LIN {X 0,Y 44.824,Z 368.173,A -85,B 0,C 180,E1 -30619.848,E2 -30619.848} C_VEL
LIN {X 0,Y 35.691,Z 373.226,A -85,B 0,C 180,E1 -30627.637,E2 -30627.637} C_VEL
LIN {X 0,Y 27.611,Z 377.135,A -85,B 0,C 180,E1 -30640.238,E2 -30640.238} C_VEL
LIN {X 0,Y 23.443,Z 379.156,A -85,B 0,C 180,E1 -30653.18,E2 -30653.18} C_VEL
LIN {X 0,Y 20.791,Z 380.755,A -85,B 0,C 180,E1 -30670.262,E2 -30670.262} C_VEL
LIN {X 0,Y 20.222,Z 381.925,A -85,B 0,C 180,E1 -30690.018,E2 -30690.018} C_VEL
LIN {X 0,Y 20.865,Z 382.602,A -85,B 0,C 180,E1 -30709.702,E2 -30709.702} C_VEL
LIN {X 0,Y 27.747,Z 382.794,A -85,B 0,C 180,E1 -30739.472,E2 -30739.472} C_VEL
LIN {X 0,Y 32.934,Z 382.312,A -85,B 0,C 180,E1 -30748.624,E2 -30748.624} C_VEL
LIN {X 0,Y 44.972,Z 380.11,A -85,B 0,C 180,E1 -30759.681,E2 -30759.681} C_VEL
LIN {X 0,Y 55.869,Z 376.992,A -85,B 0,C 180,E1 -30765.188,E2 -30765.188} C_VEL
LIN {X 0,Y 67.983,Z 372.218,A -85,B 0,C 180,E1 -30769.165,E2 -30769.165} C_VEL
LIN {X 0,Y 79.908,Z 365.993,A -85,B 0,C 180,E1 -30771.694,E2 -30771.694} C_VEL
LIN {X 0,Y 90.237,Z 359.24,A -85,B 0,C 180,E1 -30773.253,E2 -30773.253} C_VEL
LIN {X 0,Y 100.625,Z 350.879,A -85,B 0,C 180,E1 -30774.452,E2 -30774.452} C_VEL
LIN {X 0,Y 109.319,Z 342.285,A -85,B 0,C 180,E1 -30775.22,E2 -30775.22} C_VEL
LIN {X 0,Y 118.031,Z 331.706,A -85,B 0,C 180,E1 -30775.863,E2 -30775.863} C_VEL
LIN {X 0,Y 125.022,Z 321.224,A -85,B 0,C 180,E1 -30776.229,E2 -30776.229} C_VEL
LIN {X 0,Y 130.54,Z 310.906,A -85,B 0,C 180,E1 -30776.572,E2 -30776.572} C_VEL
LIN {X 0,Y 132.33,Z 306.946,A -85,B 0,C 180,E1 -30776.668,E2 -30776.668} C_VEL
LIN {X 0,Y 133.078,Z 305.198,A -85,B 0,C 180,E1 -30776.973,E2 -30776.973} C_VEL
LIN {X 0,Y 133.057,Z 305.114,A -85,B 0,C 180,E1 -30778.892,E2 -30778.892} C_VEL
LIN {X 0,Y 132.222,Z 307.019,A -85,B 0,C 180,E1 -30779.287,E2 -30779.287} C_VEL
LIN {X 0,Y 126.51,Z 318.425,A -85,B 0,C 180,E1 -30779.775,E2 -30779.775} C_VEL
LIN {X 0,Y 119.485,Z 329.469,A -85,B 0,C 180,E1 -30780.49,E2 -30780.49} C_VEL
LIN {X 0,Y 110.727,Z 340.358,A -85,B 0,C 180,E1 -30781.354,E2 -30781.354} C_VEL
LIN {X 0,Y 102.002,Z 349.18,A -85,B 0,C 180,E1 -30782.415,E2 -30782.415} C_VEL
LIN {X 0,Y 93.311,Z 356.441,A -85,B 0,C 180,E1 -30783.608,E2 -30783.608} C_VEL
LIN {X 0,Y 82.961,Z 363.561,A -85,B 0,C 180,E1 -30785.466,E2 -30785.466} C_VEL
LIN {X 0,Y 74.417,Z 368.349,A -85,B 0,C 180,E1 -30787.386,E2 -30787.386} C_VEL
LIN {X 0,Y 64.274,Z 372.98,A -85,B 0,C 180,E1 -30790.205,E2 -30790.205} C_VEL
LIN {X 0,Y 54.138,Z 376.491,A -85,B 0,C 180,E1 -30794.071,E2 -30794.071} C_VEL
LIN {X 0,Y 44.695,Z 378.993,A -85,B 0,C 180,E1 -30799.336,E2 -30799.336} C_VEL
LIN {X 0,Y 38.582,Z 380.15,A -85,B 0,C 180,E1 -30804.365,E2 -30804.365} C_VEL
LIN {X 0,Y 28.683,Z 381.121,A -85,B 0,C 180,E1 -30818.204,E2 -30818.204} C_VEL
LIN {X 0,Y 24.447,Z 381.264,A -85,B 0,C 180,E1 -30827.11,E2 -30827.11} C_VEL
LIN {X 0,Y 17.613,Z 380.911,A -85,B 0,C 180,E1 -30847.022,E2 -30847.022} C_VEL
LIN {X 0,Y 14.511,Z 380.036,A -85,B 0,C 180,E1 -30873.529,E2 -30873.529} C_VEL
LIN {X 0,Y 15.348,Z 378.997,A -85,B 0,C 180,E1 -30896.007,E2 -30896.007} C_VEL
LIN {X 0,Y 16.29,Z 378.557,A -85,B 0,C 180,E1 -30902.168,E2 -30902.168} C_VEL
LIN {X 0,Y 25.335,Z 375.258,A -85,B 0,C 180,E1 -30926.3,E2 -30926.3} C_VEL
LIN {X 0,Y 34.603,Z 371.292,A -85,B 0,C 180,E1 -30936.032,E2 -30936.032} C_VEL
LIN {X 0,Y 44.392,Z 366.186,A -85,B 0,C 180,E1 -30941.757,E2 -30941.757} C_VEL
LIN {X 0,Y 54.436,Z 359.759,A -85,B 0,C 180,E1 -30945.504,E2 -30945.504} C_VEL
LIN {X 0,Y 64.618,Z 351.765,A -85,B 0,C 180,E1 -30948.167,E2 -30948.167} C_VEL
LIN {X 0,Y 73.179,Z 343.603,A -85,B 0,C 180,E1 -30949.832,E2 -30949.832} C_VEL
LIN {X 0,Y 81.775,Z 333.642,A -85,B 0,C 180,E1 -30951.209,E2 -30951.209} C_VEL
LIN {X 0,Y 89.521,Z 322.368,A -85,B 0,C 180,E1 -30952.335,E2 -30952.335} C_VEL
LIN {X 0,Y 95.579,Z 311.302,A -85,B 0,C 180,E1 -30953.017,E2 -30953.017} C_VEL
LIN {X 0,Y 100.617,Z 299.404,A -85,B 0,C 180,E1 -30953.603,E2 -30953.603} C_VEL
LIN {X 0,Y 104.453,Z 286.706,A -85,B 0,C 180,E1 -30954.089,E2 -30954.089} C_VEL
LIN {X 0,Y 105.337,Z 282.946,A -85,B 0,C 180,E1 -30954.263,E2 -30954.263} C_VEL
LIN {X 0,Y 105.383,Z 282.402,A -85,B 0,C 180,E1 -30955.218,E2 -30955.218} C_VEL
LIN {X 0,Y 105.416,Z 282.483,A -85,B 0,C 180,E1 -30959.529,E2 -30959.529} C_VEL
LIN {X 0,Y 105.403,Z 282.822,A -85,B 0,C 180,E1 -30960.119,E2 -30960.119} C_VEL
LIN {X 0,Y 102.074,Z 295.361,A -85,B 0,C 180,E1 -30960.393,E2 -30960.393} C_VEL
LIN {X 0,Y 97.514,Z 307.417,A -85,B 0,C 180,E1 -30960.772,E2 -30960.772} C_VEL
LIN {X 0,Y 91.378,Z 319.646,A -85,B 0,C 180,E1 -30961.239,E2 -30961.239} C_VEL
LIN {X 0,Y 84.371,Z 330.532,A -85,B 0,C 180,E1 -30961.814,E2 -30961.814} C_VEL
LIN {X 0,Y 75.633,Z 341.392,A -85,B 0,C 180,E1 -30962.791,E2 -30962.791} C_VEL
LIN {X 0,Y 66.923,Z 350.211,A -85,B 0,C 180,E1 -30964.023,E2 -30964.023} C_VEL
LIN {X 0,Y 58.269,Z 357.499,A -85,B 0,C 180,E1 -30965.767,E2 -30965.767} C_VEL
LIN {X 0,Y 47.423,Z 364.989,A -85,B 0,C 180,E1 -30968.801,E2 -30968.801} C_VEL
LIN {X 0,Y 39.568,Z 369.521,A -85,B 0,C 180,E1 -30972.388,E2 -30972.388} C_VEL
LIN {X 0,Y 29.78,Z 374.22,A -85,B 0,C 180,E1 -30979.307,E2 -30979.307} C_VEL
LIN {X 0,Y 20.805,Z 377.8,A -85,B 0,C 180,E1 -30992.414,E2 -30992.414} C_VEL
LIN {X 0,Y 14.274,Z 380.367,A -85,B 0,C 180,E1 -31020.535,E2 -31020.535} C_VEL
LIN {X 0,Y 13.11,Z 381.563,A -85,B 0,C 180,E1 -31050.028,E2 -31050.028} C_VEL
LIN {X 0,Y 14.359,Z 382.256,A -85,B 0,C 180,E1 -31079.333,E2 -31079.333} C_VEL
LIN {X 0,Y 23.731,Z 382.475,A -85,B 0,C 180,E1 -31112.711,E2 -31112.711} C_VEL
LIN {X 0,Y 29.85,Z 382.013,A -85,B 0,C 180,E1 -31120.384,E2 -31120.384} C_VEL
LIN {X 0,Y 36.352,Z 381.131,A -85,B 0,C 180,E1 -31125.202,E2 -31125.202} C_VEL
LIN {X 0,Y 49.807,Z 378.168,A -85,B 0,C 180,E1 -31131.058,E2 -31131.058} C_VEL
LIN {X 0,Y 60.096,Z 374.815,A -85,B 0,C 180,E1 -31133.789,E2 -31133.789} C_VEL
LIN {X 0,Y 70.484,Z 370.408,A -85,B 0,C 180,E1 -31135.695,E2 -31135.695} C_VEL
LIN {X 0,Y 80.94,Z 364.829,A -85,B 0,C 180,E1 -31136.971,E2 -31136.971} C_VEL
LIN {X 0,Y 91.429,Z 357.889,A -85,B 0,C 180,E1 -31137.931,E2 -31137.931} C_VEL
LIN {X 0,Y 98.436,Z 352.307,A -85,B 0,C 180,E1 -31138.391,E2 -31138.391} C_VEL
LIN {X 0,Y 98.422,Z 352.302,A -85,B 0,C 180,E1 -31138.699,E2 -31138.699} C_VEL
LIN {X 0,Y 87.856,Z 360.312,A -85,B 0,C 180,E1 -31139.829,E2 -31139.829} C_VEL
LIN {X 0,Y 77.334,Z 366.711,A -85,B 0,C 180,E1 -31141.321,E2 -31141.321} C_VEL
LIN {X 0,Y 66.869,Z 371.766,A -85,B 0,C 180,E1 -31143.096,E2 -31143.096} C_VEL
LIN {X 0,Y 56.488,Z 375.674,A -85,B 0,C 180,E1 -31145.482,E2 -31145.482} C_VEL
LIN {X 0,Y 46.476,Z 378.485,A -85,B 0,C 180,E1 -31148.699,E2 -31148.699} C_VEL
LIN {X 0,Y 36.221,Z 380.432,A -85,B 0,C 180,E1 -31153.992,E2 -31153.992} C_VEL
LIN {X 0,Y 24.057,Z 381.486,A -85,B 0,C 180,E1 -31166.47,E2 -31166.47} C_VEL
LIN {X 0,Y 18.345,Z 381.46,A -85,B 0,C 180,E1 -31179.954,E2 -31179.954} C_VEL
LIN {X 0,Y 14.46,Z 381.034,A -85,B 0,C 180,E1 -31200.892,E2 -31200.892} C_VEL
LIN {X 0,Y 13.277,Z 380.188,A -85,B 0,C 180,E1 -31229.972,E2 -31229.972} C_VEL
LIN {X 0,Y 16.29,Z 378.557,A -85,B 0,C 180,E1 -31262.168,E2 -31262.168} C_VEL
LIN {X 0,Y 19.578,Z 377.263,A -85,B 0,C 180,E1 -31277.31,E2 -31277.31} C_VEL
LIN {X 0,Y 25.785,Z 374.615,A -85,B 0,C 180,E1 -31295.969,E2 -31295.969} C_VEL
LIN {X 0,Y 31.742,Z 372.046,A -85,B 0,C 180,E1 -31305.29,E2 -31305.29} C_VEL
LIN {X 0,Y 36.739,Z 369.733,A -85,B 0,C 180,E1 -31309.049,E2 -31309.049} C_VEL
LIN {X 0,Y 38.482,Z 368.857,A -85,B 0,C 180,E1 -31309.701,E2 -31309.701} C_VEL
LIN {X 0,Y 49.632,Z 362.564,A -85,B 0,C 180,E1 -31312.339,E2 -31312.339} C_VEL
LIN {X 0,Y 60.064,Z 355.193,A -85,B 0,C 180,E1 -31313.961,E2 -31313.961} C_VEL
LIN {X 0,Y 68.778,Z 347.677,A -85,B 0,C 180,E1 -31314.99,E2 -31314.99} C_VEL
LIN {X 0,Y 77.507,Z 338.575,A -85,B 0,C 180,E1 -31315.819,E2 -31315.819} C_VEL
LIN {X 0,Y 84.488,Z 329.724,A -85,B 0,C 180,E1 -31316.482,E2 -31316.482} C_VEL
LIN {X 0,Y 84.445,Z 329.802,A -85,B 0,C 180,E1 -31316.993,E2 -31316.993} C_VEL
LIN {X 0,Y 77.39,Z 338.756,A -85,B 0,C 180,E1 -31317.246,E2 -31317.246} C_VEL
LIN {X 0,Y 68.566,Z 347.964,A -85,B 0,C 180,E1 -31317.796,E2 -31317.796} C_VEL
LIN {X 0,Y 57.988,Z 356.938,A -85,B 0,C 180,E1 -31318.716,E2 -31318.716} C_VEL
LIN {X 0,Y 47.697,Z 363.989,A -85,B 0,C 180,E1 -31319.999,E2 -31319.999} C_VEL
LIN {X 0,Y 38.67,Z 369.038,A -85,B 0,C 180,E1 -31321.998,E2 -31321.998} C_VEL
LIN {X 0,Y 28.236,Z 373.772,A -85,B 0,C 180,E1 -31325.528,E2 -31325.528} C_VEL
LIN {X 0,Y 18.015,Z 377.382,A -85,B 0,C 180,E1 -31332.864,E2 -31332.864} C_VEL
LIN {X 0,Y 8.798,Z 379.979,A -85,B 0,C 180,E1 -31357.049,E2 -31357.049} C_VEL
LIN {X 0,Y 5.982,Z 381.196,A -85,B 0,C 180,E1 -31410.062,E2 -31410.062} C_VEL
LIN {X 0,Y 8.871,Z 381.911,A -85,B 0,C 180,E1 -31462.459,E2 -31462.459} C_VEL
LIN {X 0,Y 21.418,Z 382.155,A -85,B 0,C 180,E1 -31489.962,E2 -31489.962} C_VEL
LIN {X 0,Y 28.267,Z 381.711,A -85,B 0,C 180,E1 -31494.109,E2 -31494.109} C_VEL
LIN {X 0,Y 35.213,Z 380.855,A -85,B 0,C 180,E1 -31496.472,E2 -31496.472} C_VEL
LIN {X 0,Y 42.196,Z 379.585,A -85,B 0,C 180,E1 -31498.151,E2 -31498.151} C_VEL
LIN {X 0,Y 45.103,Z 378.924,A -85,B 0,C 180,E1 -31500.001,E2 -31500.001} C_VEL
LIN {X 0,Y 35.182,Z 380.71,A -85,B 0,C 180,E1 -31502.583,E2 -31502.583} C_VEL
LIN {X 0,Y 28.24,Z 381.475,A -85,B 0,C 180,E1 -31505.335,E2 -31505.335} C_VEL
LIN {X 0,Y 14.807,Z 381.793,A -85,B 0,C 180,E1 -31518.254,E2 -31518.254} C_VEL
LIN {X 0,Y 8.929,Z 381.381,A -85,B 0,C 180,E1 -31538.015,E2 -31538.015} C_VEL
LIN {X 0,Y 6.166,Z 380.562,A -85,B 0,C 180,E1 -31589.94,E2 -31589.94} C_VEL
LIN {X 0,Y 11.222,Z 378.872,A -85,B 0,C 180,E1 -31643.328,E2 -31643.328} C_VEL
LIN {X 0,Y 22.207,Z 375.68,A -85,B 0,C 180,E1 -31661.649,E2 -31661.649} C_VEL
LIN {X 0,Y 32.383,Z 371.743,A -85,B 0,C 180,E1 -31667.532,E2 -31667.532} C_VEL
LIN {X 0,Y 38.482,Z 368.857,A -85,B 0,C 180,E1 -31669.701,E2 -31669.701} C_VEL
LIN {X 0,Y 41.299,Z 370.661,A -85,B 0,C 180,E1 -31670.45,E2 -31670.45} C_VEL
LIN {X 0,Y 41.299,Z 600,A -85,B 0,C 180,E1 -31670.45,E2 -31670.45} C_VEL
LIN {X 0,Y 41.299,Z 600,A -85,B 0,C 180,E1 -31670.45,E2 -31670.45}

QRS_NEXT_CUT()

QRS_NEXT()
QRS_HOME()

END
